FUNCTION_BLOCK FB_SimulatedDigOutClose_AFO IMPLEMENTS ITF_Schuif_DigOutClose_AFO
VAR
	internalState : BOOL := FALSE;
END_VAR

{warning 'Add method implementation '}
METHOD set : BOOL
VAR_INPUT
	state : BOOL;
END_VAR
internalState := state;
END_METHOD

END_FUNCTION_BLOCK

(* stored: Version 1.1.0.1, ProductVersion 3.1.4026.8
   POU FB_SimulatedDigOutClose_AFO: Id {74c5bc87-2149-467a-b240-e636fd7104c0}, SpecialFunc None
   Method set: Id {5f1fbc6f-4731-49e0-bf19-9086eeb636a7} *)
